PROGRAM RobotDynamics

VAR
	// master robot arms joint data
	m_masterJointsData AT %I* :ST_MasterJointData;
	
	// dynamic output
	m_masterDynaData AT %Q* : ST_MasterDynaData;
	
	// flag to init robot dynamic model
	m_robotDynaInit :BOOL :=FALSE;
	
	// master grivity model 
	m_gravityModel :ARRAY[1..g_mArmNum] OF FB_MasterGravity;
	
	// master arm dynamic model
	m_armDynamic :ARRAY[1..g_mArmNum] OF FB_MasterDynamic;
	
	// master friction model
	m_frictionModel : ARRAY[1..g_mArmNum] OF FB_MasterFriciton;
	
	// master external torque observer
	m_jntDOB : ARRAY[1..g_mArmNum] OF FB_JntObserver;
	
	//master arm joint inertia
	m_jntInertia : ARRAY[1..g_mArmNum] OF FB_JntInertia;
	
	// code execute time measure
	m_codeTime : Profiler;
	
	i: INT;
	
END_VAR

m_codeTime(START:=TRUE, RESET:=TRUE);

// wait config file loaded
IF NOT(SafetyCheck.m_loadConfigFileOK) THEN
	RETURN;
END_IF

// robot dynamic model init
IF m_robotDynaInit =FALSE THEN
	FOR i:=1 TO g_mArmNum DO
		m_gravityModel[i].Init(i);
		m_armDynamic[i].init(i);
		m_frictionModel[i].init(i);
		// NOTE: curJntPos is usually zero when init, so observer need some time to stable after code run
		m_jntDOB[i].init(i, m_masterJointsData.m_curJntPos[i]); 
		m_jntInertia[i].init(i);
	END_FOR

	m_robotDynaInit:=TRUE;
END_IF

FOR i:=1 TO g_mArmNum DO
	// run gravity model
	m_gravityModel[i].run(m_masterJointsData.m_curJntPos[i], m_masterDynaData.m_gravity[i]);
	
	// run dynamic model
	m_armDynamic[i].updateDynamic(m_masterJointsData.m_curJntPos[i]);
	m_masterDynaData.m_massMat[i]:=m_armDynamic[i].jntMassMat;
	m_masterDynaData.m_lambda[i]:=m_armDynamic[i].cartMassMat;
	m_masterDynaData.m_dynaNullspace[i]:=m_armDynamic[i].dynaNullspace;
	
	// run friction model
	m_masterDynaData.m_friction[i] := m_frictionModel[i].run(m_masterDynaData.m_gravity[i],m_masterJointsData.m_curJntVel[i]);
	
(*	// run DOB
	 m_masterDynaData.m_jntExtTrq[i] := m_jntDOB[i].run(m_masterJointsData.m_curJntTrq[i], m_masterJointsData.m_curJntPos[i], m_masterDynaData.m_massMat[i]);
	// remove gravity and friction from external torque
	vecSelfAdd(m_masterDynaData.m_jntExtTrq[i], m_masterDynaData.m_gravity[i]);
	vecSelfAdd(m_masterDynaData.m_jntExtTrq[i], m_masterDynaData.m_friction[i]);*)
	
	//joint inertia torque
	m_masterDynaData.m_jntExtTrq[i]:=m_jntInertia[i].jntInertiaCal(m_masterJointsData.m_curJntPos[i],m_masterJointsData.m_curLinkPos[i],m_masterDynaData);
END_FOR

m_codeTime(START:=FALSE);

END_PROGRAM

(* stored: Version 1.1.0.1, ProductVersion 3.1.4024.11
   POU RobotDynamics: Id {798b314f-0a53-4e08-997d-5fefed426c86}, SpecialFunc None *)
